ABB RobotStudio station: FInalProject_Matos.rspag

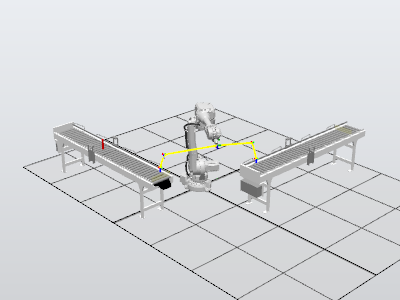
--- station ---
Station FInalProject_Matos (saved by RobotStudio 25.2.11266.1)
Controller IRB4600_45_205
  mechanical unit ROB_1: IRB4600_45_205_C_01, 6 joints, base frame (0, 0, 0) mm
Layout (positions relative to the parent item):
  - IRB4600_45_205_C_01 [mechanism, from %ABB.RobotStudio.Models.IRB4600%\IRB4600_45_205_C_G_01.rslib] at (0, 0, 0) mm; joint values [-0.5236, 0, 0, 0, 0.5236, 0] (rad or m)
  - Smart_Gripper_Servo_Fingers [mechanism] at (1084.19, -625.96, 1502.5) mm, rotated rx 180 ry 60 rz 150 deg; joint values [0.025] (rad or m)
      TCP Servo at (0, 0, 114.2) mm
      links: HandBase, DownFinger, UpFinger, VacuumOne, VacuumTwo
  - Conveyor_2 [part, from %ABB.RobotStudio.Models.Conveyors%\Conveyor Guide 400.rslib] at (1500, 0, 0) mm, rotated rx 0 ry 0 rz 90 deg
  - Conveyor_1 [part, from %ABB.RobotStudio.Models.Conveyors%\Conveyor Guide 400.rslib] at (-2500, -1500, 0) mm
  - ROD [part] at (-1200, -1300, 780) mm, size 40 x 40 x 200 mm
  - PlaneSensor [smart component, from Components\PlaneSensor.rslib]
      properties: Origin=[0.455 -1.5 0.78]; Axis1=[0 0.4 0]; Axis2=[0 0 0.1]; Tag=(none); SenseMultiple=false; SensedPart=(none)
    - _sensorPart_ [part], size 0 x 400 x 100 mm
  - Positioner [smart component, from Components\Positioner.rslib]
      properties: Object=ROD; Position=[-1.2 -1.3 0.78]; Orientation=[0 0 0]; Reference=Global; ReferenceObject=(none)
  - LinearMover [smart component, from Components\LinearMover.rslib]
      properties: Object=ROD; Direction=[1 0 0]; Speed=0.5; Reference=Global; ReferenceObject=(none)
  - LogicSRLatch [smart component, from Components\LogicSRLatch.rslib]
  - Attacher [smart component, from Components\Attacher.rslib]
      properties: Parent=Smart_Gripper_Servo_Fingers; Flange=0; Child=ROD; Mount=false; Offset=[0 0 0]; Orientation=[0 0 0]
  - Detacher [smart component, from Components\Detacher.rslib]
      properties: Child=ROD; KeepPosition=true
  - PlaneSensor_2 [smart component, from Components\PlaneSensor.rslib] at (2.31, 2137.55, 0) mm, rotated rx 0 ry 0 rz 90.41 deg
      properties: Origin=[0.451761062878983 -1.50095023240395 0.78]; Axis1=[0.00285148872345431 0.399989836135945 0]; Axis2=[0 0 0.1]; Tag=(none); SenseMultiple=false; SensedPart=(none)
    - _sensorPart_ [part], size 2.9 x 400 x 100 mm
  - LogicSRLatch_2 [smart component, from Components\LogicSRLatch.rslib]
  - LinearMover_2 [smart component, from Components\LinearMover.rslib]
      properties: Object=ROD; Direction=[0 1 0]; Speed=0.5; Reference=Global; ReferenceObject=(none)
  - LogicGate [smart component, from Components\LogicGate.rslib]
      properties: Operator=OR; Delay=0
Attachment: Smart_Gripper_Servo_Fingers is attached to IRB4600_45_205_C_01 / Link6
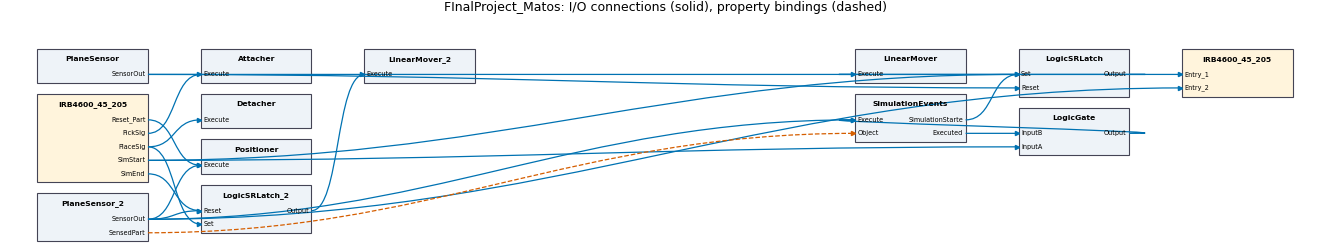
Station logic (signal -> signal, property => property):
  LogicSRLatch.Output -> LinearMover.Execute
  SimulationEvents.SimulationStarted -> LogicSRLatch.Set
  PlaneSensor.SensorOut -> LogicSRLatch.Reset
  IRB4600_45_205.Reset_Part -> Positioner.Execute
  IRB4600_45_205.PickSig -> Attacher.Execute
  IRB4600_45_205.PlaceSig -> Detacher.Execute
  PlaneSensor.SensorOut -> IRB4600_45_205.Entry_1
  PlaneSensor_2.SensorOut -> LogicSRLatch_2.Reset
  LogicSRLatch_2.Output -> LinearMover_2.Execute
  IRB4600_45_205.PlaceSig -> LogicSRLatch_2.Set
  PlaneSensor_2.SensorOut -> IRB4600_45_205.Entry_2
  PlaneSensor_2.SensorOut -> Positioner.Execute
  IRB4600_45_205.SimStart -> LogicSRLatch.Set
  IRB4600_45_205.SimEnd -> LogicSRLatch_2.Reset
  PlaneSensor_2.SensorOut -> Sink.Execute
  Sink.Executed -> LogicGate.InputB
  IRB4600_45_205.SimStart -> LogicGate.InputA
  LogicGate.Output -> Source.Execute
  PlaneSensor_2.SensedPart => Sink.Object
Targets, tools, work objects and paths stored in the station and not in the controller backup, written as RAPID:
! task T_ROB1
MODULE Module1
  PROC StopOp()
    WaitTime 2;
    Reset SimStart;
    Reset SimEnd;
    ClearVars;
  ENDPROC
  PROC RunContinous()
    ClearVars;
  ENDPROC
ENDMODULE


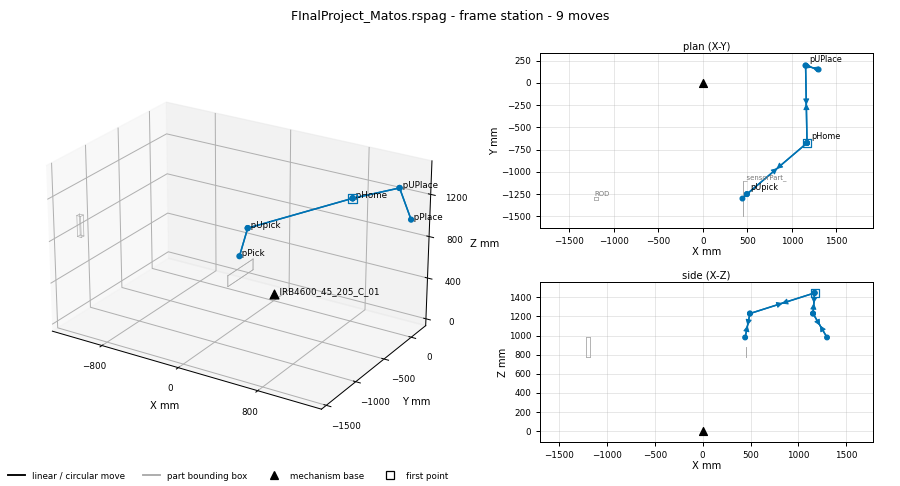
[picture p0: tool path of FInalProject_Matos.rspag in frame station, 9 of 9 moves have a stored position in this frame; points joined in program order, loops and branches not executed]
--- Controller Data/IRB4600_45_205/RAPID/TASK1/PROGMOD/CalibData.modx ---
MODULE CalibData
    PERS tooldata Servo:=[TRUE,[[0,0,114.2],[1,0,0,0]],[0.215,[8.7,12.3,49.2],[1,0,0,0],0.00021,0.00024,0.00009]];
ENDMODULE

--- Controller Data/IRB4600_45_205/RAPID/TASK1/PROGMOD/Module1.modx ---
MODULE Module1

    CONST robtarget pHome:=[[1169.838831723,-675.406764404,1445.399996856],[0.482962908,0.224143873,0.836516306,-0.129409518],[-1,-1,0,0],[9E+09,9E+09,9E+09,9E+09,9E+09,9E+09]];
    CONST robtarget pUpick:=[[494,-1250,1230],[0,0,1,0],[-1,0,-1,0],[9E+09,9E+09,9E+09,9E+09,9E+09,9E+09]];
    CONST robtarget pPick:=[[444,-1300,980],[0,0,1,0],[-1,0,-1,0],[9E+09,9E+09,9E+09,9E+09,9E+09,9E+09]];
    CONST robtarget pUPlace:=[[1153.837230719,195.293528537,1230],[0,0,1,0],[0,0,0,0],[9E+09,9E+09,9E+09,9E+09,9E+09,9E+09]];
    CONST robtarget pPlace:=[[1300,150,980],[0,0,1,0],[0,0,0,0],[9E+09,9E+09,9E+09,9E+09,9E+09,9E+09]];

    VAR num NumCycle := 0;
    VAR num OpChoice := 0;

    ! --------------------------------------------------------------

    PROC main()
        TPErase;
        WHILE TRUE DO
            TPReadFK OpChoice,
                "Select Operating Mode",
                "Run Continuous",
                "Run N Cycles",
                "Exit",
                stEmpty,
                stEmpty;

            IF OpChoice = 1 THEN
                RunContinuous;

            ELSEIF OpChoice = 2 THEN
                RunNCycles;

            ELSEIF OpChoice = 3 THEN
                TPWrite "Exiting Program.";
                RETURN;

            ELSE
                TPWrite "Invalid selection.";
            ENDIF
        ENDWHILE
    ENDPROC

    ! --------------------------------------------------------------

    PROC RunContinuous()
        TPWrite "Starting continuous run...";
        WHILE TRUE DO
            PPR;
        ENDWHILE
    ENDPROC

    ! --------------------------------------------------------------

    PROC RunNCycles()
        TPReadNum NumCycle, "Enter Desired Number of Cycles";

        FOR i FROM 1 TO NumCycle DO
            TPWrite "Cycle " + NumToStr(i,0) +
                    " of " + NumToStr(NumCycle,0);
            PPR;
        ENDFOR

        TPWrite "Completed all cycles.";
    ENDPROC

    ! --------------------------------------------------------------

    PROC PPR()
        Reset SimEnd;
        Set SimStart;
        MoveL pHome,v1000,z100,servo\WObj:=wobj0;
        WaitDI Entry_1,1;

        MoveL pUpick,v1000,z100,servo\WObj:=wobj0;
        MoveL pPick,v1000,fine,servo\WObj:=wobj0;
        WaitTime 1;
        PulseDO PickSig;
        ReSet SimStart;

        MoveL pUpick,v1000,z100,servo\WObj:=wobj0;
        MoveL pHome,v1000,z100,servo\WObj:=wobj0;

        MoveL pUPlace,v1000,z100,servo\WObj:=wobj0;
        MoveL pPlace,v1000,fine,servo\WObj:=wobj0;
        WaitTime 1;
        PulseDO PlaceSig;

        MoveL pUPlace,v1000,z100,servo\WObj:=wobj0;
        MoveL pHome,v1000,z100,servo\WObj:=wobj0;
        WaitDI Entry_2,1;
    ENDPROC

ENDMODULE

--- Controller Data/IRB4600_45_205/SYSPAR/EIO.cfg ---
EIO:CFG_1.0:7:0::
#
VIRTUAL_NETWORK:

      -Name "Virtual" -Label "Virtual Device Network"
#
EIO_SIGNAL:

      -Name "Entry_1" -SignalType "DI"

      -Name "Entry_2" -SignalType "DI"

      -Name "PickSig" -SignalType "DO" -Access "All"

      -Name "PlaceSig" -SignalType "DO" -Access "All"

      -Name "Reset_Part" -SignalType "DO" -Access "All"

      -Name "SimStart" -SignalType "DO" -Access "All"

      -Name "SimEnd" -SignalType "DO" -Access "All"

#CTRL_SIGNATURE:G01IlHOyOVAw6ccgokwxzKgZFryEi6DrPO4wxlI44hS+L/+zA11TcH/NEzMLvTyDi0gnL5Pw+rVLFXBbqg1IVQ==

--- Controller Data/IRB4600_45_205/SYSPAR/PROC.cfg ---
PROC:CFG_1.0:7:0::

#CTRL_SIGNATURE:QkSPn7KrTHat0xogrrnB9eNiUf8DpAYl1sIQTSkdl5Ic5Tdyw/+joW+l4LYglwHEvuvAgisDgbejOZqqmV6ERA==
